# EPICS substitutions: iocBoot/iocvirPV/DPU08.substitutions
file "../../db/virAi.template"{ pattern
{DPU,    num,    Temp}
{08,    0,    500}
{08,    1,    500}
{08,    2,    500}
{08,    3,    500}
{08,    4,    500}
{08,    5,    500}
{08,    6,    500}
{08,    7,    500}
{08,    8,    500}
{08,    9,    500}
{08,    10,    500}
{08,    11,    500}
{08,    12,    500}
{08,    13,    500}
{08,    14,    500}
{08,    15,    500}
{08,    16,    500}
{08,    17,    500}
{08,    18,    500}
{08,    19,    500}
{08,    20,    500}
{08,    21,    500}
{08,    22,    500}
{08,    23,    500}
{08,    24,    500}
{08,    25,    500}
{08,    26,    500}
{08,    27,    500}
{08,    28,    500}
{08,    29,    500}
{08,    30,    500}
{08,    31,    500}
{08,    32,    500}
{08,    33,    500}
{08,    34,    500}
{08,    35,    500}
{08,    36,    500}
{08,    37,    500}
{08,    38,    500}
{08,    39,    500}
{08,    40,    500}
{08,    41,    500}
{08,    42,    500}
{08,    43,    500}
{08,    44,    500}
{08,    45,    500}
{08,    46,    500}
{08,    47,    500}
{08,    48,    500}
{08,    49,    500}
{08,    50,    500}
{08,    51,    500}
{08,    52,    500}
{08,    53,    500}
{08,    54,    500}
{08,    55,    500}
{08,    56,    500}
{08,    57,    500}
{08,    58,    500}
{08,    59,    500}
{08,    60,    500}
{08,    61,    500}
{08,    62,    500}
{08,    63,    500}
{08,    64,    500}
{08,    65,    500}
{08,    66,    500}
{08,    67,    500}
{08,    68,    500}
{08,    69,    500}
{08,    70,    500}
{08,    71,    500}
{08,    72,    500}
{08,    73,    500}
{08,    74,    500}
{08,    75,    500}
{08,    76,    500}
{08,    77,    500}
{08,    78,    500}
{08,    79,    500}
{08,    80,    500}
{08,    81,    500}
{08,    82,    500}
{08,    83,    500}
{08,    84,    500}
{08,    85,    500}
{08,    86,    500}
{08,    87,    500}
{08,    88,    500}
{08,    89,    500}
{08,    90,    500}
{08,    91,    500}
{08,    92,    500}
{08,    93,    500}
{08,    94,    500}
{08,    95,    500}
{08,    96,    500}
{08,    97,    500}
{08,    98,    500}
{08,    99,    500}
{08,    100,    500}
{08,    101,    500}
{08,    102,    500}
{08,    103,    500}
{08,    104,    500}
{08,    105,    500}
{08,    106,    500}
{08,    107,    500}
{08,    108,    500}
{08,    109,    500}
{08,    110,    500}
{08,    111,    500}
{08,    112,    500}
{08,    113,    500}
{08,    114,    500}
{08,    115,    500}
{08,    116,    500}
{08,    117,    500}
{08,    118,    500}
{08,    119,    500}
{08,    120,    500}
{08,    121,    500}
{08,    122,    500}
{08,    123,    500}
{08,    124,    500}
{08,    125,    500}
{08,    126,    500}
{08,    127,    500}
{08,    128,    500}
{08,    129,    500}
{08,    130,    500}
{08,    131,    500}
{08,    132,    500}
{08,    133,    500}
{08,    134,    500}
{08,    135,    500}
{08,    136,    500}
{08,    137,    500}
{08,    138,    500}
{08,    139,    500}
{08,    140,    500}
{08,    141,    500}
{08,    142,    500}
{08,    143,    500}
{08,    144,    500}
{08,    145,    500}
{08,    146,    500}
{08,    147,    500}
{08,    148,    500}
{08,    149,    500}
{08,    150,    500}
{08,    151,    500}
{08,    152,    500}
{08,    153,    500}
{08,    154,    500}
{08,    155,    500}
{08,    156,    500}
{08,    157,    500}
{08,    158,    500}
{08,    159,    500}
{08,    160,    500}
{08,    161,    500}
{08,    162,    500}
{08,    163,    500}
{08,    164,    500}
{08,    165,    500}
{08,    166,    500}
{08,    167,    500}
{08,    168,    500}
{08,    169,    500}
{08,    170,    500}
{08,    171,    500}
{08,    172,    500}
{08,    173,    500}
{08,    174,    500}
{08,    175,    500}
{08,    176,    500}
{08,    177,    500}
{08,    178,    500}
{08,    179,    500}
{08,    180,    500}
{08,    181,    500}
{08,    182,    500}
{08,    183,    500}
{08,    184,    500}
{08,    185,    500}
{08,    186,    500}
{08,    187,    500}
{08,    188,    500}
{08,    189,    500}
{08,    190,    500}
{08,    191,    500}
{08,    192,    500}
{08,    193,    500}
{08,    194,    500}
{08,    195,    500}
{08,    196,    500}
{08,    197,    500}
{08,    198,    500}
{08,    199,    500}
}
